FUNCTION_BLOCK EBMaster (* Service Interface Function Block Type *)
  (* Description: Copyright (c) 2016 fortiss GmbH This program and the accompanying materials are made available under the terms of the Eclipse Public License 2.0 which is available at https://www.eclipse.org/legal/epl-2.0/ SPDX-License-Identifier: EPL-2.0 *)
  (* Version 3.0, 2025-04-14, Patrick Aigner, changed package *)
  (* Version 1.0, 2016-11-30, Johannes Messmer, fortiss GmbH *)
  PACKAGE eclipse4diac::io::embrick;
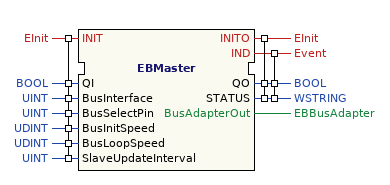
  EVENT_INPUT
    INIT : EInit WITH QI, BusInitSpeed, SlaveUpdateInterval, BusLoopSpeed, BusInterface, BusSelectPin; (* Service Initialization *)
  END_EVENT
  EVENT_OUTPUT
    INITO : EInit WITH QO, STATUS; (* Initialization Confirm *)
    IND WITH QO, STATUS; (* Indication from Resource *)
  END_EVENT
  VAR_INPUT
    QI : BOOL; (* Event Input Qualifier *)
    BusInterface : UINT := 1; (* ID of SPI interface *)
    BusSelectPin : UINT := 49; (* SPI slave select pin *)
    BusInitSpeed : UDINT := 300000; (* SPI speed during initialization *)
    BusLoopSpeed : UDINT := 700000; (* SPI speed during runtime *)
    SlaveUpdateInterval : UINT := 25; (* Global update interval of slave modules in Hz *)
  END_VAR
  VAR_OUTPUT
    QO : BOOL; (* Event Output Qualifier *)
    STATUS : WSTRING; (* Service Status *)
  END_VAR
  PLUGS
    BusAdapterOut : eclipse4diac::io::embrick::EBBusAdapter;
  END_PLUGS
END_FUNCTION_BLOCK
